DATA_BLOCK "dbArchiveAutoBoiler"
{ S7_Optimized_Access := 'TRUE' }
VERSION : 0.8
NON_RETAIN
"fbArchiveAutoBoiler"

BEGIN

END_DATA_BLOCK

